//This function is used to calculate the blade angle of each in a pair of blades, based on a symetric gap size
FUNCTION_BLOCK FB_CalculateAngle

VAR_INPUT
GapSize : LREAL;
BladeSize : LREAL;
ClosedGap : LREAL;

END_VAR

VAR_OUTPUT
AngleBladeA : LREAL;
AngleBladeB : LREAL;

END_VAR

VAR

//BLADESIZE : LREAL:=62.94;	
//CLOSEDGAP : LREAL:=2.00;

END_VAR

IF GapSize<ClosedGap THEN
    AngleBladeA:=0;
    AngleBladeB:=0;
ELSIF GapSize > (2*BladeSize+ClosedGap) THEN
    AngleBladeA:=90;
    AngleBladeB:=90;
ELSE
    AngleBladeA := RAD_TO_DEG(ACOS((BladeSize + (ClosedGap/2) - (GapSize/2))/BladeSize));
    AngleBladeB := RAD_TO_DEG(-ACOS((BladeSize + (ClosedGap/2) - (GapSize/2))/BladeSize));  
END_IF

END_FUNCTION_BLOCK

(* stored: Version 1.1.0.1, ProductVersion 3.1.4024.0
   POU FB_CalculateAngle: Id {389ded1b-c11c-4aa1-9e95-096a9e4789a7}, SpecialFunc None *)
